INTERFACE I_Cyl_AtHome

PROPERTY P_AtHome : BOOL
GET
END_GET
END_PROPERTY

END_INTERFACE

(* stored: Version 1.1.0.1, ProductVersion 3.1.4024.6
   Itf I_Cyl_AtHome: Id {4629e0ed-ef4c-0c3e-1d93-c1d7972dc166}
   Property P_AtHome: Id {a032ec04-c8a7-0225-18d5-cd8c516ff1fd}
   Get Get: Id {9d785874-7d94-0740-2ad0-6853787a57e2} *)
